{attribute 'qualified_only'}
{attribute 'strict'}
{attribute 'to_string'}
TYPE COMPARISION_RESULT :
(
	LEFT_LESS_RIGHT := -1,
	EQUALS := 0,
	LEFT_GREATER_RIGHT := 1
) SINT;
END_TYPE

(* stored: Version 1.1.0.1
   DUT COMPARISION_RESULT: Id {7e63b84a-5e8a-4ed0-a28f-03c78265f8d0} *)
